SUBAPPLICATION RedGreenBackground1_aux (* Hintergrundfarbe (TRUE -> Rot, FALSE -> Grün) für 1 Objekt *)
  (* Standard: 61499-2 *)
  (* Version 1.0, 2026-07-21, franz, Meisterschulen am Ostbahnhof *)
  PACKAGE MyLib::sys;
  IMPORT isobus::UT::Q::const::IDs::ID_NULL;
  IMPORT isobus::UT::Q::const::colours;
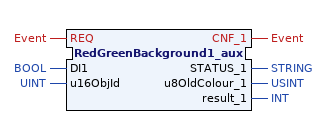
  EVENT_INPUT
    REQ; (* Normal Execution Request *)
  END_EVENT
  EVENT_OUTPUT
    CNF_1; (* Execution Confirmation *)
  END_EVENT
  VAR_INPUT
    DI1 : BOOL; (* Selector *)
    u16ObjId : UINT := ID_NULL; (* Object ID Softkey *)
  END_VAR
  VAR_OUTPUT
    STATUS_1 : STRING; (* Service Status *)
    u8OldColour_1 : USINT; (* Old value of ID *)
    result_1 : INT; (* retval see description *)
  END_VAR
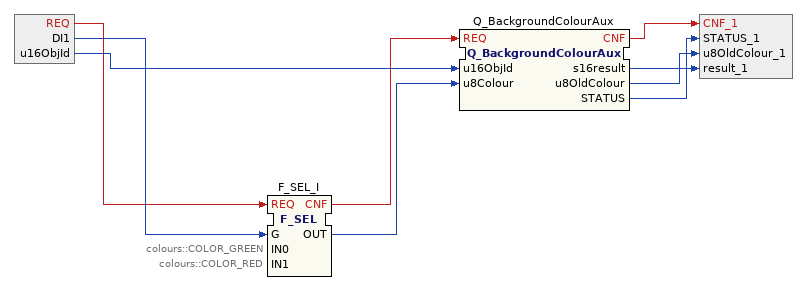
  FBS
    Q_BackgroundColourAux : isobus::UT::Q::Q_BackgroundColourAux;
    F_SEL_I : iec61131::selection::F_SEL(IN0 := colours::COLOR_GREEN, IN1 := colours::COLOR_RED);
  END_FBS
  EVENT_CONNECTIONS
    Q_BackgroundColourAux.CNF TO CNF_1;
    F_SEL_I.CNF TO Q_BackgroundColourAux.REQ;
    REQ TO F_SEL_I.REQ;
  END_CONNECTIONS
  DATA_CONNECTIONS
    u16ObjId TO Q_BackgroundColourAux.u16ObjId;
    Q_BackgroundColourAux.s16result TO result_1;
    Q_BackgroundColourAux.u8OldColour TO u8OldColour_1;
    Q_BackgroundColourAux.STATUS TO STATUS_1;
    F_SEL_I.OUT TO Q_BackgroundColourAux.u8Colour;
    DI1 TO F_SEL_I.G;
  END_CONNECTIONS
END_SUBAPPLICATION
